// Struckig
// Copyright (C) 2022 Stefan Besler

// This program is free software: you can redistribute it and/or modify
// it under the terms of the GNU General Public License as published by
// the Free Software Foundation, either version 3 of the License, or
// (at your option) any later version.

// This program is distributed in the hope that it will be useful,
// but WITHOUT ANY WARRANTY; without even the implied warranty of
// MERCHANTABILITY or FITNESS FOR A PARTICULAR PURPOSE.  See the
// GNU General Public License for more details.
//
// You should have received a copy of the GNU General Public License
// along with THIS PROGRAM.  IF NOT, see <http://www.gnu.org/licenses/>.
{attribute 'hide'}
/// Internal bit-cast helper from raw IEEE-754 bits to `LREAL`.
FUNCTION LrealFromBits : LREAL
VAR_INPUT
  b : ULINT; //< Raw floating-point bit pattern.
END_VAR
VAR
  x : POINTER TO LREAL := ADR(b);
END_VAR

LrealFromBits := x^;

END_FUNCTION

(* stored: Version 1.1.0.1
   POU LrealFromBits: Id {26af1350-f1f7-4775-a258-be47fc01563f}, SpecialFunc None *)
